// TIA Portal project "Smart Temaprature Control System Using RTD, PLC, VFD and Actuator" (V18)

(* hardware
DEVICE "S7-1200 station_1"  S7-1200 Station
   slot 0: "Rack_0"  S7-1200 Rack  Rack  V1.0
   slot 1: "PLC_1"  CPU 1215C DC/DC/DC  6ES7 215-1AG40-0XB0  V4.2
DEVICE "HMI_1"  KTP400 Basic PN
   slot 0: "HMI_1"  KTP400 Basic PN  6AV2 123-2DB03-0AX0  17.0.0.0
   slot 1: "HMI_RT_1"  KTP400 Basic PN  6AV2 123-2DB03-0AX0  17.0.0.0
   slot 5: "HMI_1.IE_CP_1"  PROFINET Interface  17.0.0.0
      slot 1: "PROFINET Interface_1"  PROFINET Interface
         slot 1: "Port_1"  Port
*)

// ===== PLC "PLC_1"  CPU 1215C DC/DC/DC =====

VAR_GLOBAL   // PLC tag table "Default tag table"
   "Tag_1" AT %MD10 : DWord;
   "Temp_out" AT %MD14 : DInt;
   "Temp Out for Real number" AT %MD18 : Real;
   "Tag_2" AT %MD22 : DWord;
   "Tag_3" AT %IW66 : Word;
   "Tag_4" AT %MD40 : Real;
   "Actuator Feedback" AT %MD44 : DInt;
   "Actuator Feedback Volt" AT %MD48 : DInt;
END_VAR

VAR_GLOBAL   // PLC tag table "System Memory"
   "Sys_memory" AT %M100.0 : Bool;
END_VAR

VAR_GLOBAL   // PLC tag table "Outputs"
   "Green_led" AT %Q0.0 : Bool;
   "Red_led" AT %Q0.1 : Bool;
   "Led_1" AT %Q0.2 : Bool;
   "Led_2" AT %Q0.3 : Bool;
   "30 HZ" AT %Q0.4 : Bool;
   "40 Hz" AT %Q0.5 : Bool;
   "Cooling Motor" AT %Q0.6 : Bool;
   "Actuator" AT %QW64 : Int;
END_VAR

VAR_GLOBAL   // PLC tag table "Inputs"
   "Stop Button" AT %I0.0 : Bool;
   "Start Button" AT %I0.1 : Bool;
   "RTD_ Temparature sensor" AT %IW64 : Int;
END_VAR

VAR_GLOBAL   // PLC tag table "HMI tags"
   "Start Button For HMI" AT %M0.0 : Bool;
   "Stop Button for HMI" AT %M0.1 : Bool;
END_VAR

ORGANIZATION_BLOCK "Main"   // OB1, LAD, ProgramCycle
TITLE = "Main Program Sweep (Cycle)"
{ S7_Optimized_Access := 'TRUE' }
VERSION : 0.1
   VAR_INPUT
      Initial_Call : Bool;   // Initial call of this OB
      Remanence : Bool;   // =True, if remanent data are available
   END_VAR
BEGIN

REGION Network 1
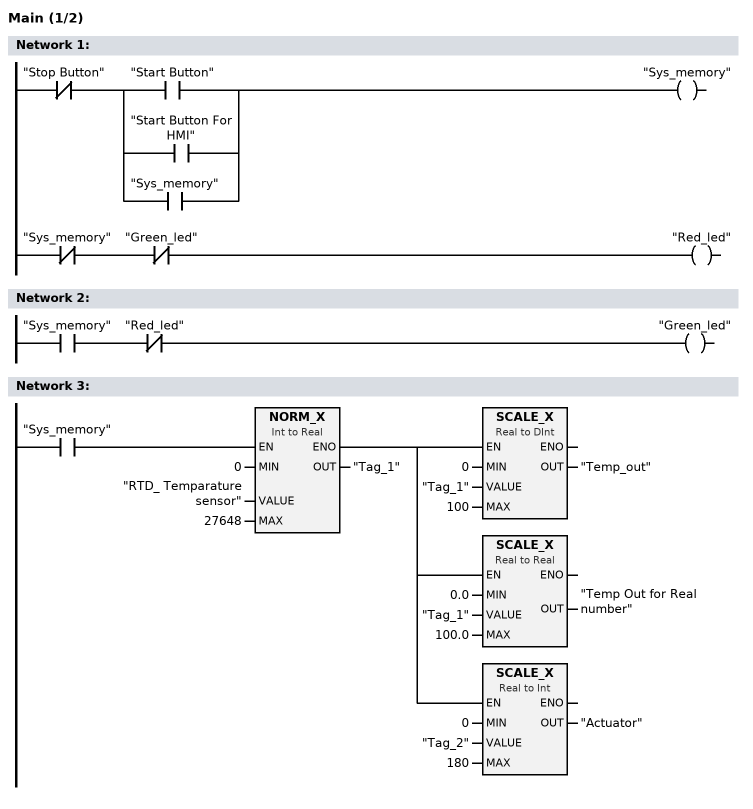
   RUNG wire#powerrail
      I_Contact( "Stop Button" )
      wire#w1
      Contact( "Start Button" )
      wire#w2
      Coil( "Sys_memory" )
   END_RUNG
   RUNG wire#w1
      Contact( "Start Button For HMI" )
   END_RUNG wire#w2
   RUNG wire#w1
      Contact( "Sys_memory" )
   END_RUNG wire#w2
   RUNG wire#powerrail
      I_Contact( "Sys_memory" )
      I_Contact( "Green_led" )
      Coil( "Red_led" )
   END_RUNG
   // the same network as SCL:
   "Sys_memory" := NOT "Stop Button" AND ("Start Button" OR "Start Button For HMI" OR "Sys_memory");
   "Red_led" := NOT "Sys_memory" AND NOT "Green_led";
END_REGION

REGION Network 2
   RUNG wire#powerrail
      Contact( "Sys_memory" )
      I_Contact( "Red_led" )
      Coil( "Green_led" )
   END_RUNG
   // the same network as SCL:
   "Green_led" := "Sys_memory" AND NOT "Red_led";
END_REGION

REGION Network 3
   RUNG wire#powerrail
      Contact( "Sys_memory" )
      { S7_Templates := "[SrcType := Int, DestType := Real]" } Normalize(min := 0, value := "RTD_ Temparature sensor", max := 27648, out => "Tag_1")
      wire#w1
      { S7_Templates := "[SrcType := Real, DestType := DInt]" } Scale(min := 0, value := "Tag_1", max := 100, out => "Temp_out")
   END_RUNG
   RUNG wire#w1
      { S7_Templates := "[SrcType := Real, DestType := Real]" } Scale(min := 0.0, value := "Tag_1", max := 100.0, out => "Temp Out for Real number")
   END_RUNG
   RUNG wire#w1
      { S7_Templates := "[SrcType := Real, DestType := Int]" } Scale(min := 0, value := "Tag_2", max := 180, out => "Actuator")
   END_RUNG
   // the same network as SCL:
   IF "Sys_memory" THEN
       "Tag_1" := NORM_X(MIN := 0, VALUE := "RTD_ Temparature sensor", MAX := 27648);
       "Temp_out" := SCALE_X(MIN := 0, VALUE := "Tag_1", MAX := 100);
       "Temp Out for Real number" := SCALE_X(MIN := 0.0, VALUE := "Tag_1", MAX := 100.0);
       "Actuator" := SCALE_X(MIN := 0, VALUE := "Tag_2", MAX := 180);
   END_IF;
END_REGION

REGION Network 4
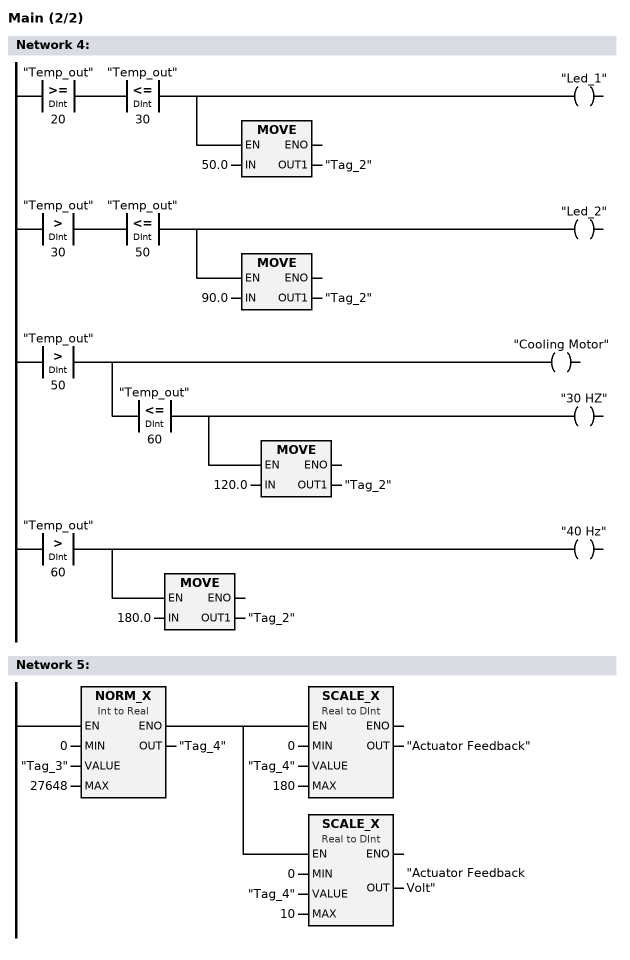
   RUNG wire#powerrail
      { S7_Templates := "SrcType := DInt" } GE_Contact(in1 := "Temp_out", in2 := 20)
      { S7_Templates := "SrcType := DInt" } LE_Contact(in1 := "Temp_out", in2 := 30)
      wire#w1
      Coil( "Led_1" )
   END_RUNG
   RUNG wire#w1
      Move(in := 50.0, out1 => "Tag_2")
   END_RUNG
   RUNG wire#powerrail
      { S7_Templates := "SrcType := DInt" } GT_Contact(in1 := "Temp_out", in2 := 30)
      { S7_Templates := "SrcType := DInt" } LE_Contact(in1 := "Temp_out", in2 := 50)
      wire#w2
      Coil( "Led_2" )
   END_RUNG
   RUNG wire#w2
      Move(in := 90.0, out1 => "Tag_2")
   END_RUNG
   RUNG wire#powerrail
      { S7_Templates := "SrcType := DInt" } GT_Contact(in1 := "Temp_out", in2 := 50)
      wire#w3
      Coil( "Cooling Motor" )
   END_RUNG
   RUNG wire#w3
      { S7_Templates := "SrcType := DInt" } LE_Contact(in1 := "Temp_out", in2 := 60)
      wire#w4
      Coil( "30 HZ" )
   END_RUNG
   RUNG wire#w4
      Move(in := 120.0, out1 => "Tag_2")
   END_RUNG
   RUNG wire#powerrail
      { S7_Templates := "SrcType := DInt" } GT_Contact(in1 := "Temp_out", in2 := 60)
      wire#w5
      Coil( "40 Hz" )
   END_RUNG
   RUNG wire#w5
      Move(in := 180.0, out1 => "Tag_2")
   END_RUNG
   // the same network as SCL:
   "Led_1" := ("Temp_out" >= 20) AND ("Temp_out" <= 30);
   IF "Led_1" THEN "Tag_2" := 50.0; END_IF;
   "Led_2" := ("Temp_out" > 30) AND ("Temp_out" <= 50);
   IF "Led_2" THEN "Tag_2" := 90.0; END_IF;
   "Cooling Motor" := "Temp_out" > 50;
   "30 HZ" := "Cooling Motor" AND ("Temp_out" <= 60);
   IF "30 HZ" THEN "Tag_2" := 120.0; END_IF;
   "40 Hz" := "Temp_out" > 60;
   IF "40 Hz" THEN "Tag_2" := 180.0; END_IF;
END_REGION

REGION Network 5
   RUNG wire#powerrail
      { S7_Templates := "[SrcType := Int, DestType := Real]" } Normalize(min := 0, value := "Tag_3", max := 27648, out => "Tag_4")
      wire#w1
      { S7_Templates := "[SrcType := Real, DestType := DInt]" } Scale(min := 0, value := "Tag_4", max := 180, out => "Actuator Feedback")
   END_RUNG
   RUNG wire#w1
      { S7_Templates := "[SrcType := Real, DestType := DInt]" } Scale(min := 0, value := "Tag_4", max := 10, out => "Actuator Feedback Volt")
   END_RUNG
   // the same network as SCL:
   "Tag_4" := NORM_X(MIN := 0, VALUE := "Tag_3", MAX := 27648);
   "Actuator Feedback" := SCALE_X(MIN := 0, VALUE := "Tag_4", MAX := 180);
   "Actuator Feedback Volt" := SCALE_X(MIN := 0, VALUE := "Tag_4", MAX := 10);
END_REGION
END_ORGANIZATION_BLOCK

(* ===== HMI "HMI_RT_1" =====
system functions are stored by id; their names below are inferred from use
connection "HMI_Connection_1": ETHERNET, SMART_S7_1200_OMS

HMI tags "Default tag table"
   "Tag_ScreenNumber" : UInt, internal
   "Start Button For HMI" : Bool = PLC "Start Button For HMI" AT %M0.0, 1 s
   "Stop Button for HMI" : Bool = PLC "Stop Button for HMI" AT %M0.1, 1 s
   "Green_led" : Bool = PLC Green_led AT %Q0.0, 1 s
   "Red_led" : Bool = PLC Red_led AT %Q0.1, 1 s
   "Cooling Motor" : Bool = PLC "Cooling Motor" AT %Q0.6, 1 s
   "Led_1" : Bool = PLC Led_1 AT %Q0.2, 1 s
   "Led_2" : Bool = PLC Led_2 AT %Q0.3, 1 s
   "30 HZ" : Bool = PLC "30 HZ" AT %Q0.4, 1 s
   "40 Hz" : Bool = PLC "40 Hz" AT %Q0.5, 1 s
   "Temp Out for Real number" : Real = PLC "Temp Out for Real number" AT %MD18, 1 s
   "Actuator Feedback Volt" : DInt = PLC "Actuator Feedback Volt" AT %MD48, 1 s
   "Actuator Feedback" : DInt = PLC "Actuator Feedback" AT %MD44, 1 s
   "Sys_memory" : Bool = PLC Sys_memory AT %M100.0, 1 s
   "Temp_out" : DInt = PLC Temp_out AT %MD14, 1 s

text list "System": 0 'System OFF'; 1 'System ON'

text list "C. Motor": 0 'C. Motor OFF'; 1 'C. Motor ON'

graphic list "Motor": 0 'Graphic_3'; 1 'Graphic_4'

screen "Root screen" 480x272, template "Template_1"
   on GenerateScreen: SetTag("Tag_ScreenNumber", 1)
   Button "Button_1" at 21,25 size 101x49; TextOff 'Start'
      on Press: function_b14e0dd5("Start Button For HMI", 0)
   Button "Button_2" at 19,91 size 103x47; TextOff 'Stop'
      on Press: function_b14e0dd5("Stop Button for HMI", 0)
   Circle "Circle_1" at 214,12 size 48x48
      Appearance <- "Green_led"
   TextField "Text field_1" at 201,65 size 71x20; Text 'GREEN LED'
   Circle "Circle_2" at 305,12 size 48x48
      Appearance <- "Red_led"
   TextField "Text field_2" at 292,65 size 57x20; Text 'RED LED'
   Circle "Circle_3" at 396,12 size 48x48
      Appearance <- "Cooling Motor"
   TextField "Text field_3" at 396,63 size 44x20; Text 'Motor'
   Circle "Circle_4" at 183,108 size 48x48
      Appearance <- "Led_1"
   TextField "Text field_4" at 189,156 size 42x20; Text 'LED-1'
   Circle "Circle_5" at 255,108 size 48x48
      Appearance <- "Led_2"
   TextField "Text field_5" at 261,156 size 42x20; Text 'LED-2'
   Circle "Circle_6" at 324,108 size 48x48
      Appearance <- "30 HZ"
   TextField "Text field_6" at 324,156 size 41x20; Text '30 HZ'
   Circle "Circle_7" at 392,108 size 48x48
      Appearance <- "40 Hz"
   TextField "Text field_7" at 392,156 size 41x20; Text '40 HZ'
   IOField "I/O field_2" at 25,185 size 84x39; FormatPattern 999
      ProcessValue <- "Temp_out"
   IOField "I/O field_1" at 181,183 size 84x40; FormatPattern 999
      ProcessValue <- "Actuator Feedback"
   IOField "I/O field_3" at 349,185 size 84x39; FormatPattern 999
      ProcessValue <- "Actuator Feedback Volt"
   TextField "Text field_8" at 25,223 size 70x20; Text 'Temp_Out'
   TextField "Text field_9" at 141,218 size 153x20; Text 'Actuator Feedback (D)'
   TextField "Text field_10" at 317,225 size 153x20; Text 'Actuator Feedback (V)'
   Button "Button_3" at 183,240 size 96x32; TextOff 'Next Screen'
      on Click: ActivateScreen("Next Screen", 0)

screen "Next Screen" 480x272
   SymbolicIOField "Symbolic I/O field_1" at 0,0 size 118x50; TextOff '0'; TextOn '1'; TextList "System"
      ProcessValue <- "Sys_memory"
   SymbolicIOField "Symbolic I/O field_2" at 0,69 size 118x47; TextOff '0'; TextOn '1'; TextList "C. Motor"
      ProcessValue <- "Cooling Motor"
   GraphicIOField "Graphic I/O field_1" at 233,66 size 76x60; PictureList "Motor"
      ProcessValue <- "Cooling Motor"
   Bar "Bar_1" at 400,2 size 80x269; MinimumValue 0; MaximumValue 100
      ProcessValue <- "Temp_out"
   Button "Button_1" at 167,251 size 2x0; TextOff 'Text'
   Button "Button_2" at 185,240 size 96x32; TextOff 'Back'
      on Click: ActivateScreen("Root screen", 0)
*)